Staubli VAL3: GETVALUE.pgx

public program getValue(bool x_bUseLatch, num& x_nEncValue[])
begin
  // This routine returns either the latched or the actual value
  // of the encoder
  //
  // Input Param
  //  xUseLatch define which kind of encoder value should be returned
  //    x_bUseLatch=true --> returns the value of the Latch register
  //    x_bUseLatch=false--> returns the current of the counter.
  //
  // Output Param
  //  x_nEncValue : Encoder value
  //
  // Created 23-02-05                                   C.CURRIVAND
  //----------------------------------------------------------------
  if x_bUseLatch==true
    x_nEncValue=nEncLatchedVal
  else
    x_nEncValue=nEncValue
  endIf
end
